// TIA Portal V20 export
FUNCTION_BLOCK "GM_SendFData"   // FB23, LAD
TITLE = Template: GM sending data
// Template v0.1
// stored: MemoryReserve 100, Namespace Safety, SetENOAutomatically false
   VAR_INPUT
      Connection_ID_Send : Word;
      Connection_ID_Receive : Word;
   END_VAR
   VAR_IN_OUT
      Send_Array : Array[0..121] of Byte;
      Receive_Ack_Send_Array : Array[0..21] of Byte;
   END_VAR
   VAR
      instTSendData : TSEND;   // Send data to PLC 2
      instTSendAck { S7_SetPoint := 'True'} : TSEND;   // Send acknowledge data to PLC 2
      statErrorSendData { S7_SetPoint := 'True'} : Word;   // variable for saving the status of TSEND block in case of error
      statErrorSendAck : Word;   // variable for saving the status of TSEND block in case of error
      statSendTimer { S7_SetPoint := 'True'} : TON_TIME;   // SendAckScanD/T
   END_VAR
   VAR_TEMP   // added for the SCL form of the ladder/FBD networks
      _w1 : Bool;
   END_VAR
BEGIN

REGION Network 1: Send F-Data to PLC2 / Send F-data to partner
   // Sending F-data by calling TSEND-Block with REQ = 0 first and REQ = 1 afterwards to ensure positive edge on REQ in order to send it on each cycle.
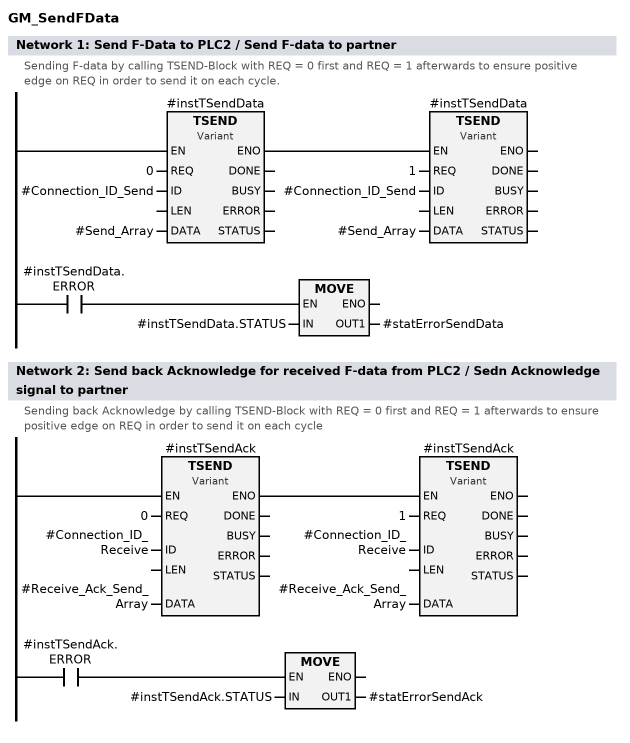
   RUNG wire#powerrail
      { S7_Templates := "[data_type := Variant, len_type := UDInt, id_type := CONN_OUC]" } #instTSendData.TSEND(REQ := 0, ID := #Connection_ID_Send, LEN :=, DATA := #Send_Array, DONE =>, BUSY =>, ERROR =>, STATUS =>)
      { S7_Templates := "[data_type := Variant, len_type := UDInt, id_type := CONN_OUC]" } #instTSendData.TSEND(REQ := 1, ID := #Connection_ID_Send, LEN :=, DATA := #Send_Array, DONE =>, BUSY =>, ERROR =>, STATUS =>)
   END_RUNG
   RUNG wire#powerrail
      Contact( #instTSendData.ERROR )
      Move(in := #instTSendData.STATUS, out1 => #statErrorSendData)
   END_RUNG
   // the same network as SCL:
   #instTSendData(REQ := 0, ID := #Connection_ID_Send, DATA := #Send_Array, ENO => #_w1);   // TSEND
   IF #_w1 THEN
       #instTSendData(REQ := 1, ID := #Connection_ID_Send, DATA := #Send_Array);   // TSEND
   END_IF;
   IF #instTSendData.ERROR THEN #statErrorSendData := #instTSendData.STATUS; END_IF;
END_REGION

REGION Network 2: Send back Acknowledge for received F-data from PLC2 / Sedn Acknowledge signal to partner
   // Sending back Acknowledge by calling TSEND-Block with REQ = 0 first and REQ = 1 afterwards to ensure positive edge on REQ in order to send it on each cycle
   RUNG wire#powerrail
      { S7_Templates := "[data_type := Variant, len_type := UDInt, id_type := CONN_OUC]" } #instTSendAck.TSEND(REQ := 0, ID := #Connection_ID_Receive, LEN :=, DATA := #Receive_Ack_Send_Array, DONE =>, BUSY =>, ERROR =>, STATUS =>)
      { S7_Templates := "[data_type := Variant, len_type := UDInt, id_type := CONN_OUC]" } #instTSendAck.TSEND(REQ := 1, ID := #Connection_ID_Receive, LEN :=, DATA := #Receive_Ack_Send_Array, DONE =>, BUSY =>, ERROR =>, STATUS =>)
   END_RUNG
   RUNG wire#powerrail
      Contact( #instTSendAck.ERROR )
      Move(in := #instTSendAck.STATUS, out1 => #statErrorSendAck)
   END_RUNG
   // the same network as SCL:
   #instTSendAck(REQ := 0, ID := #Connection_ID_Receive, DATA := #Receive_Ack_Send_Array, ENO => #_w1);   // TSEND
   IF #_w1 THEN
       #instTSendAck(REQ := 1, ID := #Connection_ID_Receive, DATA := #Receive_Ack_Send_Array);   // TSEND
   END_IF;
   IF #instTSendAck.ERROR THEN #statErrorSendAck := #instTSendAck.STATUS; END_IF;
END_REGION
END_FUNCTION_BLOCK
